(* IEC 61131-3 sources: CodesysTest/alpha/export/Device.dev/Plc Logic/Application, 4 files *)

(* ---- Globals.gvl.st ---- *)
(*#-#-#-#-#-#-#-#-#-#---Declaration---#-#-#-#-#-#-#-#-#-#-#-#-#*)

{attribute 'qualified_only'}
VAR_GLOBAL
    firstScan : BOOL; //First Scan Bit
    pressureBarServoCommsType : MODBUS_COMM_TYPE;  //Comm path to Pressure Bar Servo - 0 = TCP, 1 = RTU
    STEPS_PER_INCH : INT;  //Steps Per Inch for Pressure Bar Servos
    enableDryCycle : BOOL;          // Enable dry cycle
	SystemLog : FB_InternalLogger;
	jawMovingIn : BOOL;
	passthroughChangedFromJog : BOOL;
	machinePowerOK : BOOL;
END_VAR

VAR_GLOBAL CONSTANT
    STEPS_PER_INCH_SEAL_FLATTENER_HORIZONTAL_AXIS_MOTOR  : INT := 2500;
    STEPS_PER_INCH_SEAL_FLATTENER_VERTICAL_AXIS_MOTOR : INT := 2890;        //Steps per inch for NEMA 17 seal flattener finger motor
    STEPS_PER_INCH_BIG_MOTOR : INT := 21872;        //Steps per inch for NEMA 17 motor
    STEPS_PER_INCH_SMALL_MOTOR : INT := 19600;        //Steps per inch for NEMA 11 motor
    STEPS_PER_INCH_SHOW_MOTOR : INT := 18900;        //Steps per inch for NEMA 11 motor
    STEPS_PER_INCH_PRINTER : INT := 4498;            //Steps per inch for printer step servo
    STEPS_PER_INCH_20_DEGREE_BAG_DELIVERY : INT := 5093; // Steps per inch for 20 degree bag delivery motors
	STEPS_PER_INCH_PRO24_BAG_DELIVERY : INT := 4428; // Steps per inch for 20 degree bag delivery motors
	STEPS_PER_INCH_ADJUSTABLE_PASSTHROUGH : INT := 3030;  // Steps per inch for the Adjustable Passthrough motor
	STEPS_PER_INCH_TFBelt : INT := 3030;  // Steps per inch for the Adjustable Passthrough motor
	STEPS_PER_INCH_TFLS : INT := 10000;  // Steps per inch for the Adjustable Passthrough motor
    VELOCITY_IPS_MULTIPLIER_20_DEGREE_BAG_DELIVERY: REAL := 53;
    PASSTHROUGH_ZERO_OFFSET : REAL := 2;            //Zero offset for passthough (minimum passthough)
    MAX_BAG_WIDTH : REAL := 18;                //Passthrough setting
	AMP_MOTOR_RPI : INT := 10;
	MAX_LOGGED_ITEMS : UINT := 500;	// Max items to be logged
END_VAR

VAR_GLOBAL
    headCycleCount : DINT;                 // Head Cycle Counts
	headCycleCount2 : DINT;                 // Head Cycle Counts
    bagGrabberCycleCount : DINT;         // Bag Grabber Cycle Counts
    solenoidCycleCount1 : DINT;         // Solenoid Cycle Cycle Counts (first solenoid)
    motorizedSealFlattenersCount : DINT;         // MSF Cycle Counts
    bagOpenFingersCount : DINT;        // Bag Open Finger Cycles
    sealFlattenerFingersCount : DINT;  // Seal Flattener Fingers Cycle Count
    electricPressureBarCount : DINT;    // Electric Pressure bar Cycle count
    sealBarCount : DINT;                 // Seal bar Cycle count
    bagDeliveryCycleCount : DINT;        // Bag Delivery Cycle Count
    printerCycleCounts : DINT;            // Printer Cycle Counts
    bagsMadeCount : DINT;                // Bags Made
    passthroughChangeCount : DINT;        // Passthrough Changes
	passthroughChangeDistance : UDINT;	// Passthrough Distance Changes in .1 Inches
	solenoidCycleCount2 : DINT;     	// Solenoid Cycle Cycle Counts (Strech SX)
	solenoidFailureCount2 : UDINT;		// Solenoid Failure Count (Strech SX)
	pickAndPlaceCycleCount : UDINT;		// Pick and place cycle count
	passthroughChangeCount2 : DINT;        // Passthrough Changes
	passthroughChangeDistance2 : UDINT;	// Passthrough Distance Changes in .1 Inches
	bagFailedToGrabBothFingersCount : UDINT; // Both Fingers failed to grab bag
	bagFailedToGrabRightFingerCount : UDINT; // Right Bag Open Finger Failed to Grab Bag
	bagFailedToGrabLeftFingerCount : UDINT; // Left Bag Open Finger Failed to Grab Bag
	successfulBagOpenCount : UDINT;			// Successful Bag Open Count
	rejectedBagCount : UDINT;				// Rejected bag count
    dryCycleCount  :UDINT;                   // Dry cycle count
	lastPrinterDelta : TIME := T#100MS;
	factoryTestComplete : BOOL;		// 1000 bags test done
END_VAR

(* ---- HMIData.gvl.st ---- *)
(*#-#-#-#-#-#-#-#-#-#---Declaration---#-#-#-#-#-#-#-#-#-#-#-#-#*)

// All HMI data is presented through this GVL
{attribute 'qualified_only'}
{attribute 'global_init_slot' := '50001'}
VAR_GLOBAL //PERSISTENT RETAIN
	initiateCycle : BOOL;  // Initiate Cycle Pushbutton
	ackAllFaults : BOOL; // Acknowledge All Faults from HMI
	makeReady : BOOL;
	jobLoaded : BOOL;
    stopMachine : BOOL;
	version : STRING;
	inCycle : BOOL;
	batchEnable : BOOL;
	batchSetting : UDINT := 10;
	batchCount : UDINT;
	headCycleCount : UDINT;
	pressureBarOpenDelay : REAL;
	pressureBarCloseDelay : REAL;
	passthroughSetting : REAL := 5.0;
	passthroughOffset : REAL;
	passthroughPosition : REAL;
	lpaDwell : REAL;
	hpaDwell : REAL;
	sealBarDwell : REAL;
	sealBarTemperatureSetting : UDINT;
	sealBarTemperature : UDINT;
	sealFlattenersPosition : REAL;
	bagSkirtLength : REAL := 1.35;
	bagLength : REAL := 23.5;
	bagWidth : REAL := 17.5;
	bagThickness : REAL := 2.5;
	bagTensionSetting : REAL := 0.6;  // Bag takeup tension setting in amps
	bagDropTime : REAL;
	bagForwardSpeed : UDINT := 55;
	bagReverseSpeed : UDINT := 3;
	bagEdgePhotoeyeCovered : BOOL;
	printSpeed : UDINT := 6;
	printLength : REAL := 8.0;
	printOffset : REAL := 2.0;
	fillerCountSetting : UDINT;
	fillerCurrentCount : UDINT;
	fillerDropTime : REAL;
	loadPlateDelay : REAL;
	loadPlateDwell : REAL;
	exitConveyorDwell : REAL;
	vacuumDwell : REAL := 0.25;
	IBDDeflateDwellTime  : REAL := 0.75;
	IBDPackageEjectAssistDelayTime : REAL;
	IBDPackageEjectAssistDwellTime : REAL := 0.8;
	funnelInUse : BOOL;								// Funnel Enable/Disable
	funnelOpenDelay : REAL := 0.25;					// Funnel Open Delay after pressure bar open
	funnelOpeningTime : REAL := 0.5;				// For funnel w/o sensors only : Time required to consider funnel open after command to open
	funnelClosingTime : REAL := 0.5;				// For funnel w/o sensors only : Time required to consider funnel closed after command to close
	externalExitConveyorDwell : REAL;
	barcodeGoodReadCount : UDINT;
	barcodeBadReadCount : UDINT;
	barcodeBadReadFaultSetting : UDINT;
	barcodeStartPosition : REAL;
	barcodeScanDistance : REAL := 1.0;
	barcodeVerifierInUse : BOOL;
	barcodeLastReadString : STRING[100];
	lastCycleTime : REAL;
	averageCycleTime : REAL;
	resetAverageCycleTime : BOOL;
	bagOpenRetrySetting : INT := 3;
	bagOpenRetryCount : INT;
	bagOpenFeedNewBagSetting : INT := 1;
	bagOpenFeedNewBagCount : INT;
	currentJobID : INT;
	separateBeforeSeal : BOOL;
	activateDemoMode : BOOL;
	printerInUse : BOOL;
	printerInstalled : BOOL;
	lpaDuringBagFeedEnable : BOOL := TRUE;
	lpaBagEjectAssistEnable : BOOL := TRUE;

	(*Service Stuff*)
	lpaServiceOn : BOOL;
	lpaServiceOff : BOOL;
	lpaServicePulse : BOOL;
	hpaServiceOn :BOOL;
	hpaServicePulse : BOOL;
	exitConveyorStart : BOOL;
	exitConveyorStop : BOOL;
	exitConveyorJog : BOOL;
	exitConveyorJogTime : TIME;
	exitConveyorStartDwell : BOOL;
	pressureBarService : ServiceCommands;
	loadPlateService : ServiceCommands;
	forwardLoadPlateService : ServiceCommands;
	rearLoadPlateService : ServiceCommands;
	loadShelfService : ServiceCommands;
	IBDService : ServiceCommands;
	funnelService : ServiceCommands;
	baggerHeadService : ServiceCommands;
	jogBagForward : BOOL;
	jogBagReverse : BOOL;
	jogPassthroughForward : BOOL;
	jogPassthroughReverse : BOOL;
	sealBarServiceCycle : BOOL;
	sealBarServiceRetract : BOOL;
	sealBarServiceExtend : BOOL;
	bagOpenFingersServiceGrab : BOOL;
	bagOpenFingersServiceRelease : BOOL;
	sealFlattenersServiceRaise : BOOL;
	sealFlattenersServiceLower : BOOL;
	sealFlattenersServiceJogIn : BOOL;
	sealFlattenersServiceJogOut : BOOL;
	sealFlattenersManualPositionSetting : REAL;
	sealFlattenersMoveToManualPos : BOOL;
	passthroughManualPositionSetting : REAL;
	passthroughMoveToManualPos : BOOL;
	factoryTestMode : BOOL;
	vacuumServiceOn : BOOL;
	vacuumServiceOff : BOOL;
	printHeadServiceRaise : BOOL;
	printHeadServiceLower : BOOL;
	externalExitConveyorStart : BOOL;
	externalExitConveyorStop : BOOL;
	externalExitConveyorJog : BOOL;
	externalExitConveyorStartDwell : BOOL;
	triggerBarcodeReaderService : BOOL;

	(*Factoy Config*)
	bofSelection : BagOpenFingersSelection := BagOpenFingersSelection.PneumaticWithBagOpenSensors;
	sealFlattenersSelection : SealFlattenerSelection := SealFlattenerSelection.MotorizedSealFlatteners;
	printerSelection : LabelPrinterSelection := LabelPrinterSelection.ZebraPrinter203DPI;
	integratedExitConveyorSelection : IntegratedConveyorSelection := IntegratedConveyorSelection.RearExit;
	externalExitConveyorSelection : ExteralConveyorSelection := ExteralConveyorSelection.NotInstalled;
	packageEjectSelection : PackageEjectionSelection := PackageEjectionSelection.RearRetractingLoadPlate;
	independentBagDeflatorSelection : BagDeflatorSelection := BagDeflatorSelection.NotInstalled;
	cycleStartButtonSelection : PalmButtonSelection := PalmButtonSelection.DualPalmButton;
	barcodeVerifierSelection : BCVSelection := BCVSelection.NotInstalled;
	baggerModelSelection : ModelSelection;
	auxIOConfig : AuxIOConfiguration;
	fillerFactorySelection : FillerSelection;
	funnelFactorySelection : FunnelSelection;
	murrIOConfigVersion : CONFIG_VERSIONS := CONFIG_VERSIONS.V_1_4;
	printerConfigVersion : CONFIG_VERSIONS := CONFIG_VERSIONS.V_1_2;
	frontFilmFeedMotorConfigVersion : CONFIG_VERSIONS := CONFIG_VERSIONS.V_1_0;
	rearUnwindMotorConfigVersion : CONFIG_VERSIONS := CONFIG_VERSIONS.V_1_1;
	sealFlattenerMotorConfigVersion : CONFIG_VERSIONS := CONFIG_VERSIONS.V_1_0;

	(*Warnings*)
	printerRibbonLow : Warning;
	printerNotReady : Warning;
	waitingForPrinter : Warning;
	sealBarNotAtTemperature : Warning;
	recoveryModeActive : Warning;
	jobLoadRequired : Warning;
	baggerNotReady : Warning;
	demoModeIsActive : Warning;
	factoryTestModeActive : Warning;
	machineNotTested : Warning;
	packageEjectGuardRemoved : Warning;
	bagLevelLow : Warning;
	fillerModeCycleStartOnly : Warning;
	baggerInhibited : Warning;
	(*Misc*)
	pressureBarState : STRING;

    (*Counters*)
    baggerCycles : FB_CycleCounter;
	bagOpenFingerCycles : FB_CycleCounter;
	bagsMade : FB_CycleCounter;
	sealBarCycles : FB_CycleCounter;
	pressureBarCycles : FB_CycleCounter;
	passthroughChanges : FB_CycleCounter;
	loadPlateCycles : FB_CycleCounter;
	printerCycles : FB_CycleCounter;
	motorizedSealFlattenerCycles : FB_CycleCounter;
	bagOpenRetryTotal : FB_CycleCounter;
	bagsRejectedTotal : FB_CycleCounter;
	resettableBagsMade : FB_CycleCounter;

	(*Predictive Maint.*)
	airFilterClean : FB_PredictiveMaint := (target := 30000, count := 0, name := 'Clean Air Filter');
	driveRollerClean : FB_PredictiveMaint := (target := 20000, count := 0, name := 'Clean Drive Rollers', units := 'Inches of Bag');
	printHeadClean : FB_PredictiveMaint := (target := 10000, count := 0, name := 'Clean Print Head', units := 'Printer Cycles');
	pressureBarGuideShaftGuides : FB_PredictiveMaint := (target := 0, count := 127888, name := 'Replace Guide Shafts');

	pressureBarLeak : FB_CylinderLeak := (maximumStrokeTime := 5.0, name := 'Pressure Bar Stroke', units := 'Seconds');
	loadPlateLeak : FB_CylinderLeak := (maximumStrokeTime := 2.0, name := 'Load Plate Stroke', units := 'Seconds');

	msfHorizontalMotorTemp : FB_DriveTemp := (maxTemp := 60.0, name := 'MSF Motor Temp.', units := 'deg C');
	bagDeliveryMotorTemp : FB_DriveTemp := (maxTemp := 60.0, name := 'Bag Delivery Motor Temp.', units := 'deg C');
	passthroughMotorTemp : FB_DriveTemp := (maxTemp := 60.0, name := 'Passthrough Motor Temp.', units := 'deg C');

	(*Info*)
	faultActive : BOOL;

END_VAR

VAR_GLOBAL CONSTANT
	murrIOConfigVersionMax : CONFIG_VERSIONS := CONFIG_VERSIONS.V_1_4;
	printerConfigVersionMax : CONFIG_VERSIONS := CONFIG_VERSIONS.V_1_2;
	frontFilmFeedMotorConfigVersionMax : CONFIG_VERSIONS := CONFIG_VERSIONS.V_1_0;
	rearUnwindMotorConfigVersionMax : CONFIG_VERSIONS := CONFIG_VERSIONS.V_1_1;
	sealFlattenerMotorConfigVersionMax : CONFIG_VERSIONS := CONFIG_VERSIONS.V_1_0;
END_VAR

(* ---- RecallValues.pou.st ---- *)
(*#-#-#-#-#-#-#-#-#-#---Declaration---#-#-#-#-#-#-#-#-#-#-#-#-#*)

FUNCTION RecallValues : DWORD
VAR
	recipieManager : Recipe_Management.RecipeManCommands;
	recipeName : STRING;
	recResult : DWORD;
END_VAR
(*#-#-#-#-#-#-#-#-#-#---Implementation---#-#-#-#-#-#-#-#-#-#-#-#-#*)

recResult := recipieManager.GetRecipeNames('Recipes', ADR(recipeName),1,0);
recResult := recipieManager.LoadAndWriteRecipe(RecipeDefinitionName := 'Recipes', RecipeName := recipeName);

(* ---- SaveValues.pou.st ---- *)
(*#-#-#-#-#-#-#-#-#-#---Declaration---#-#-#-#-#-#-#-#-#-#-#-#-#*)

FUNCTION SaveValues : DWORD
VAR
	recipieManager : Recipe_Management.RecipeManCommands;
	recipeName : STRING;
	recResult : DWORD;
END_VAR
(*#-#-#-#-#-#-#-#-#-#---Implementation---#-#-#-#-#-#-#-#-#-#-#-#-#*)

//IF HMIData.bagsMade.count <> 0 THEN
	recResult := recipieManager.CreateRecipe(RecipeDefinitionName := 'Recipes', RecipeName := 'Automatic');
	recResult := recipieManager.GetRecipeNames('Recipes', ADR(recipeName),1,0);
	recResult := recipieManager.ReadAndSaveRecipe(RecipeDefinitionName := 'Recipes', RecipeName := recipeName);
//END_IF
